// SIMATIC S7-200 project (STEP 7-Micro/WIN), CPU 224XP REL 02.01

SYMBOL_TABLE 用户定义1
TJBZW            M0.3     // 停机标志位
TJ               Q0.7     // 停机
DJD              I0.1     // 电接点压力低
YLD              T45      // 压力低延时
YJQT             I0.5     // 一键启停
GZSC             Q0.5     // 故障输出
ZSGG             M0.1     // 转速过高标志位
Jiansu           Q0.3     // 减速
ZDTS             M0.5     // 自动提速
QDCG             M0.0     // 启动成功位
GF               Q0.6     // 关阀
FMKDW            I0.3     // 阀门开到位
KF               Q0.2     // 开阀
JS               Q0.1     // 加速
YLDXH            M10.0    // 压力低标志位
ZD               I0.0     // 自动
ZDTR             Q0.4     // 自动投入指示
TZ               M10.3    // 停止位
QD               M10.2    // 启动位
END_SYMBOL_TABLE

ORGANIZATION_BLOCK 主程序:OB1
TITLE=程序注释
BEGIN
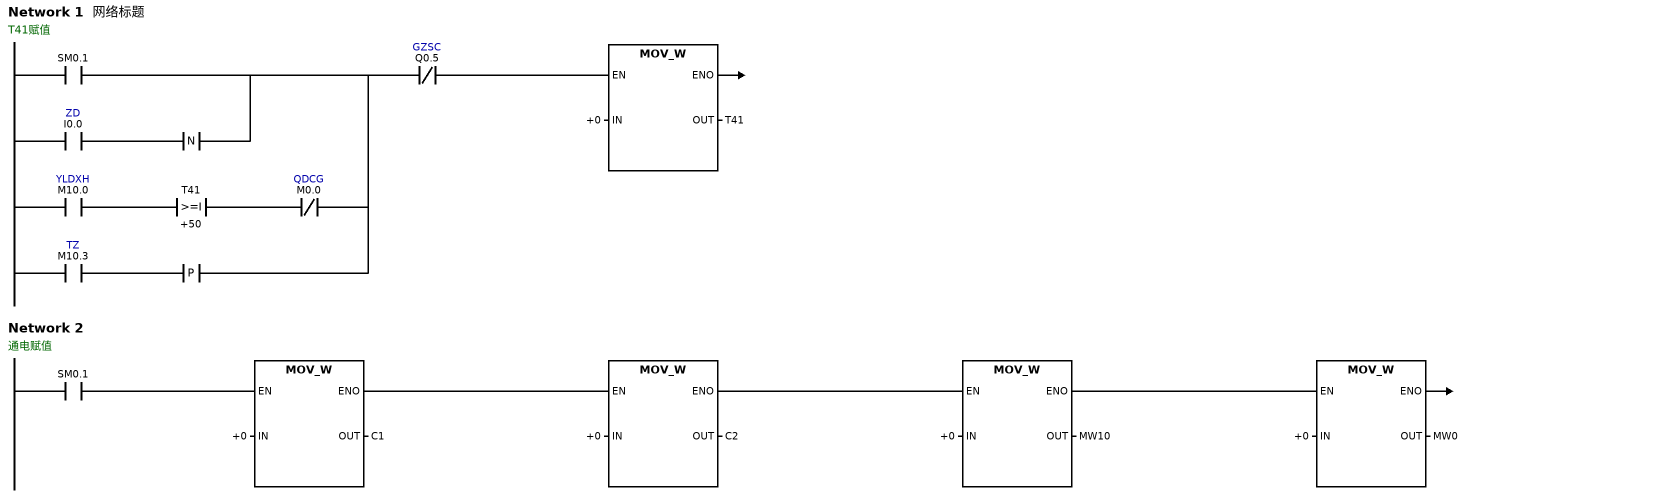
Network 1 // 网络标题
// T41赋值
LD     SM0.1
LD     ZD:I0.0
ED
OLD
LD     YLDXH:M10.0
AW>=   T41, +50
AN     QDCG:M0.0
OLD
LD     TZ:M10.3
EU
OLD
AN     GZSC:Q0.5
MOVW   +0, T41
Network 2
// 通电赋值
LD     SM0.1
MOVW   +0, C1
AENO
MOVW   +0, C2
AENO
MOVW   +0, MW10
AENO
MOVW   +0, MW0
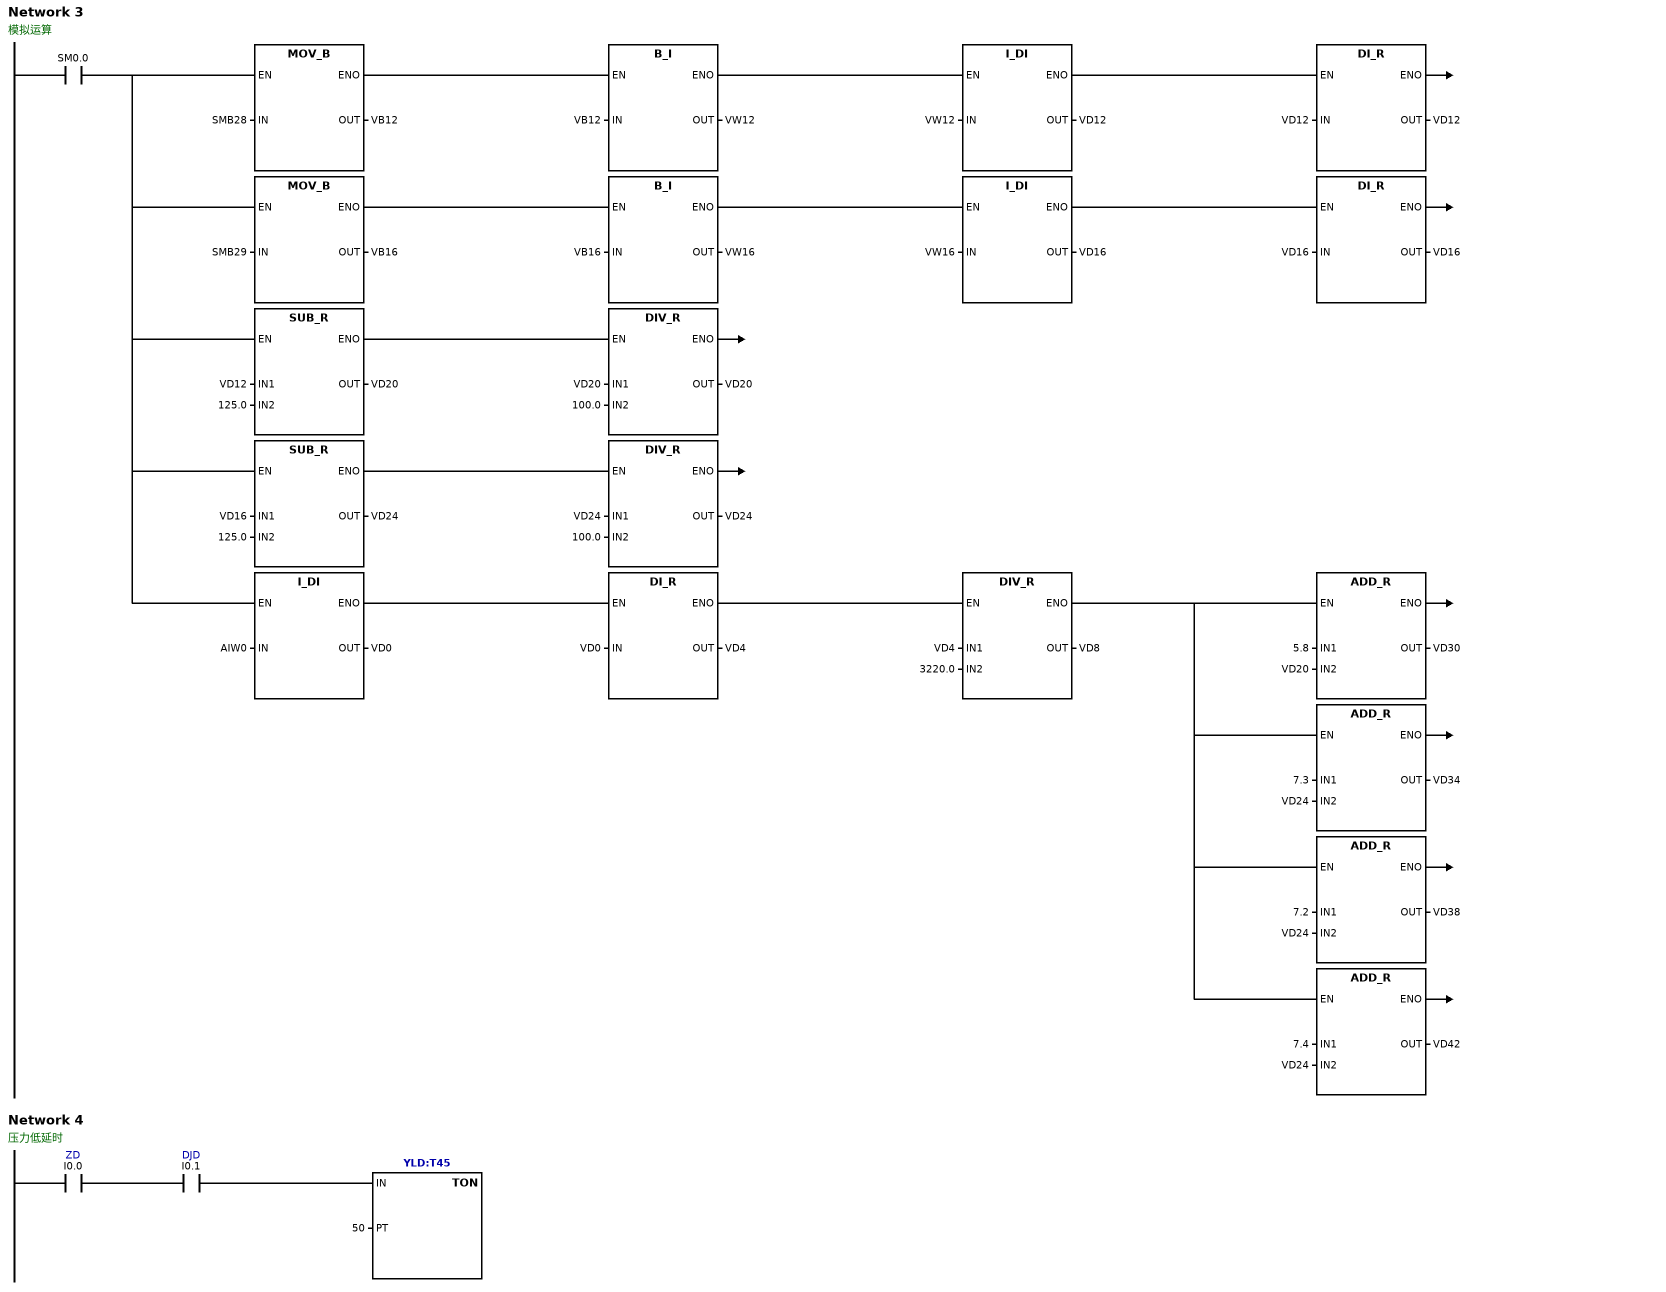
Network 3
// 模拟运算
LD     SM0.0
LPS
MOVB   SMB28, VB12
AENO
BTI    VB12, VW12
AENO
ITD    VW12, VD12
AENO
DTR    VD12, VD12
LRD
MOVB   SMB29, VB16
AENO
BTI    VB16, VW16
AENO
ITD    VW16, VD16
AENO
DTR    VD16, VD16
LRD
MOVR   VD12, VD20
AENO
-R     125.0, VD20
AENO
/R     100.0, VD20
LRD
MOVR   VD16, VD24
AENO
-R     125.0, VD24
AENO
/R     100.0, VD24
LPP
ITD    AIW0, VD0
AENO
DTR    VD0, VD4
AENO
MOVR   VD4, VD8
AENO
/R     3220.0, VD8
AENO
MOVR   5.8, VD30
+R     VD20, VD30
MOVR   7.3, VD34
+R     VD24, VD34
MOVR   7.2, VD38
+R     VD24, VD38
MOVR   7.4, VD42
+R     VD24, VD42
Network 4
// 压力低延时
// (network saved uncompiled; LAD cells follow)
// row 0: c0 -| |- ZD:I0.0  c1 -| |- DJD:I0.1  c2 --  c3 [TON YLD:T45 IN:=power@row0, PT:=50]
// row 1: c3 [box]
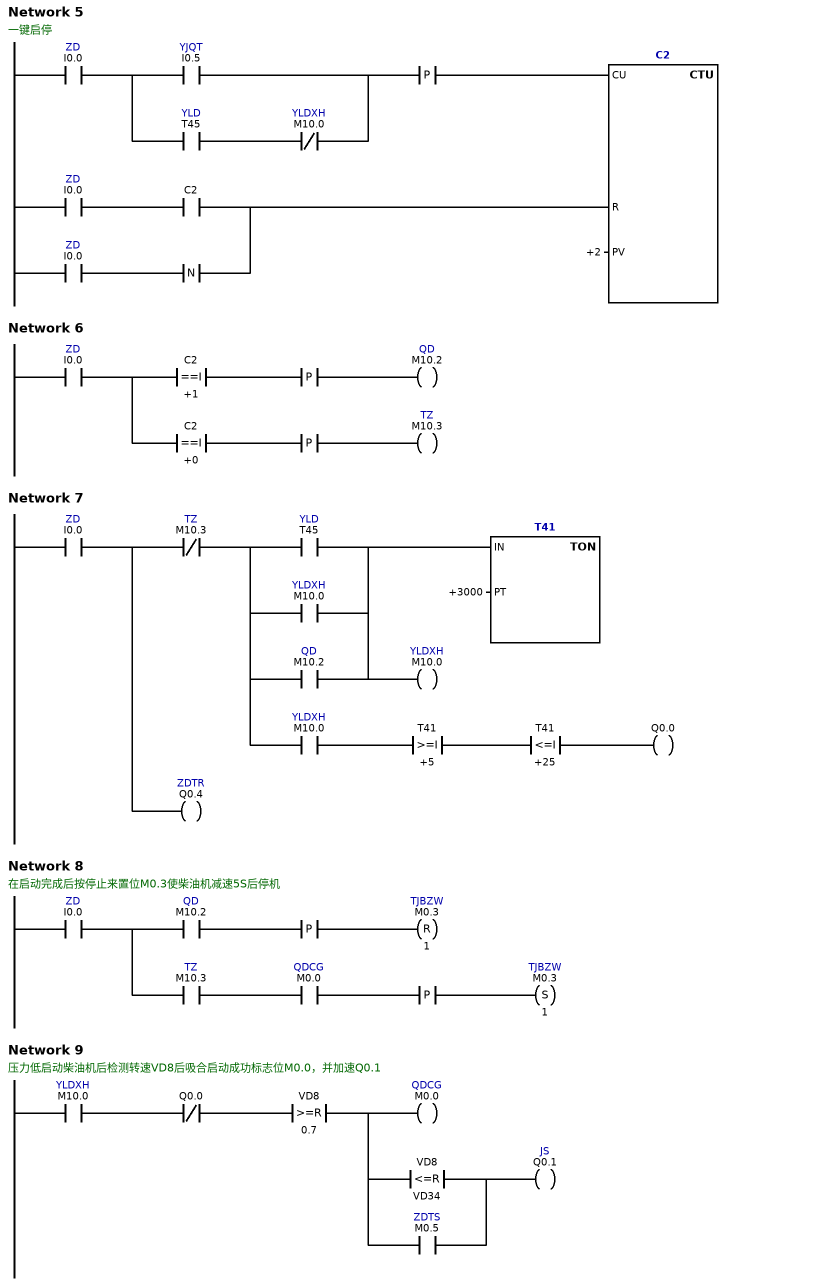
Network 5
// 一键启停
// (network saved uncompiled; LAD cells follow)
// row 0: c0 -| |- ZD:I0.0 v  c1 -| |- YJQT:I0.5  c2 -- v  c3 -|P|-  c4 --  c5 [CTU C2 CU:=power@row0, R:=power@row2, PV:=+2]
// row 1: c0 ^  c1 -| |- YLD:T45  c2 -|/|- YLDXH:M10.0 ^  c5 [box]
// row 2: c0 -| |- ZD:I0.0  c1 -| |- C2 v  c2 --  c3 --  c4 --  c5 [box]
// row 3: c0 -| |- ZD:I0.0  c1 -|N|-  ^  c5 [box]
Network 6
LD     ZD:I0.0
LPS
AW=    C2, +1
EU
=      QD:M10.2
LPP
AW=    C2, +0
EU
=      TZ:M10.3
Network 7
LD     ZD:I0.0
LPS
AN     TZ:M10.3
LPS
LD     YLD:T45
O      YLDXH:M10.0
O      QD:M10.2
ALD
TON    T41, +3000
=      YLDXH:M10.0
LPP
A      YLDXH:M10.0
AW>=   T41, +5
AW<=   T41, +25
=      Q0.0
LPP
=      ZDTR:Q0.4
Network 8
// 在启动完成后按停止来置位M0.3使柴油机减速5S后停机
// (network saved uncompiled; LAD cells follow)
// row 0: c0 -| |- ZD:I0.0 v  c1 -| |- QD:M10.2  c2 -|P|-  c3 -(R) TJBZW:M0.3, 1
// row 1: c0 ^  c1 -| |- TZ:M10.3  c2 -| |- QDCG:M0.0  c3 -|P|-  c4 -(S) TJBZW:M0.3, 1
Network 9
// 压力低启动柴油机后检测转速VD8后吸合启动成功标志位M0.0，并加速Q0.1
LD     YLDXH:M10.0
AN     Q0.0
AR>=   VD8, 0.7
=      QDCG:M0.0
LDR<=  VD8, VD34
O      ZDTS:M0.5
ALD
=      JS:Q0.1
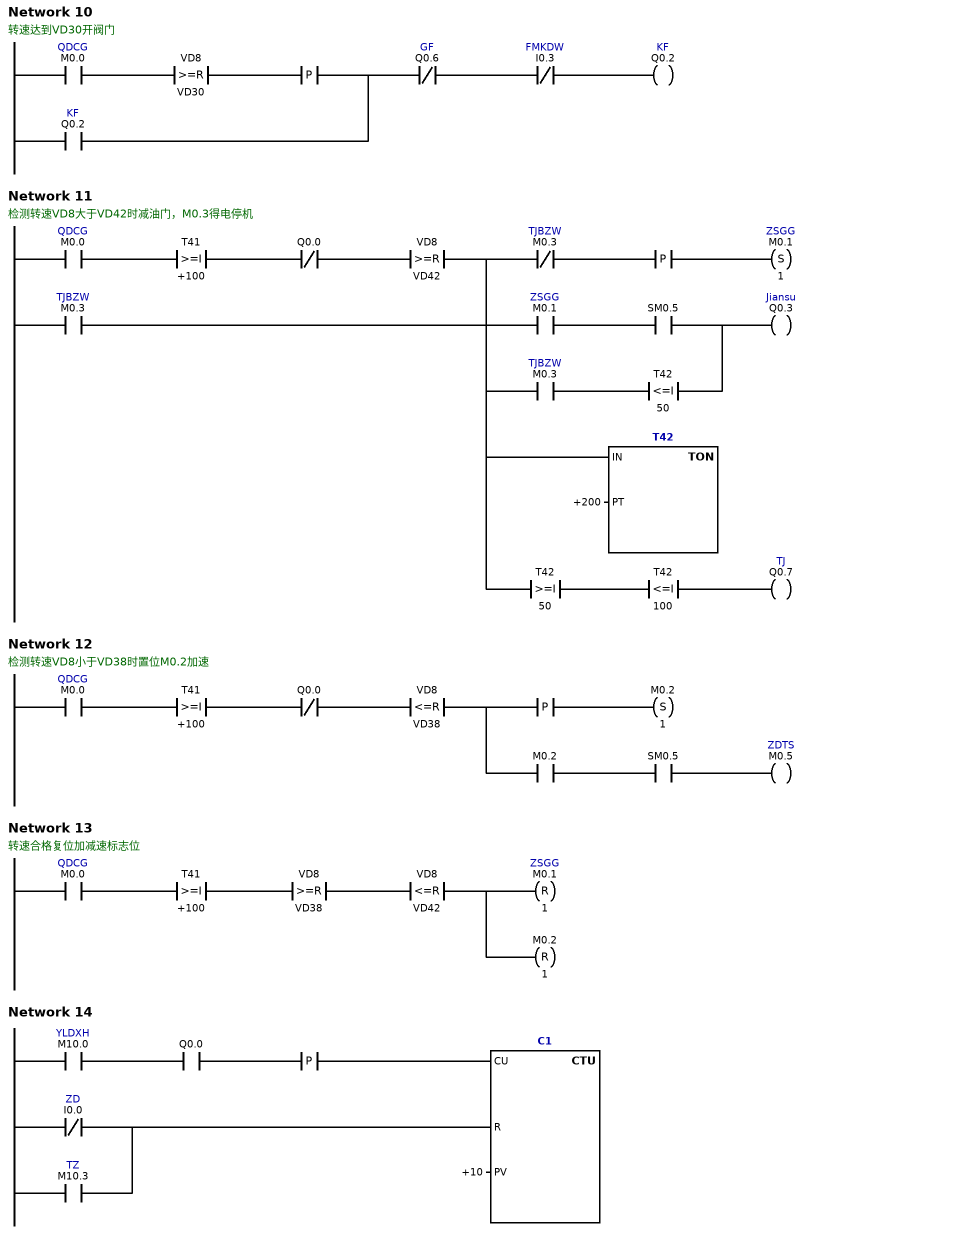
Network 10
// 转速达到VD30开阀门
LD     QDCG:M0.0
AR>=   VD8, VD30
EU
O      KF:Q0.2
AN     GF:Q0.6
AN     FMKDW:I0.3
=      KF:Q0.2
Network 11
// 检测转速VD8大于VD42时减油门，M0.3得电停机
// (network saved uncompiled; LAD cells follow)
// row 0: c0 -| |- QDCG:M0.0  c1 -|>=I|- T41, +100  c2 -|/|- Q0.0  c3 -|>=R|- VD8, VD42 v  c4 -|/|- TJBZW:M0.3  c5 -|P|-  c6 -(S) ZSGG:M0.1, 1
// row 1: c0 -| |- TJBZW:M0.3  c1 --  c2 --  c3 -- ^v  c4 -| |- ZSGG:M0.1  c5 -| |- SM0.5 v  c6 -( ) Jiansu:Q0.3
// row 2: c3 ^v  c4 -| |- TJBZW:M0.3  c5 -|<=I|- T42, 50 ^
// row 3: c3 ^v  c4 --  c5 [TON T42 IN:=power@row3, PT:=+200]
// row 4: c3 ^v  c5 [box]
// row 5: c3 ^  c4 -|>=I|- T42, 50  c5 -|<=I|- T42, 100  c6 -( ) TJ:Q0.7
Network 12
// 检测转速VD8小于VD38时置位M0.2加速
LD     QDCG:M0.0
AW>=   T41, +100
AN     Q0.0
AR<=   VD8, VD38
LPS
EU
S      M0.2, 1
LPP
A      M0.2
A      SM0.5
=      ZDTS:M0.5
Network 13
// 转速合格复位加减速标志位
LD     QDCG:M0.0
AW>=   T41, +100
AR>=   VD8, VD38
AR<=   VD8, VD42
R      ZSGG:M0.1, 1
R      M0.2, 1
Network 14
LD     YLDXH:M10.0
A      Q0.0
EU
LDN    ZD:I0.0
O      TZ:M10.3
CTU    C1, +10
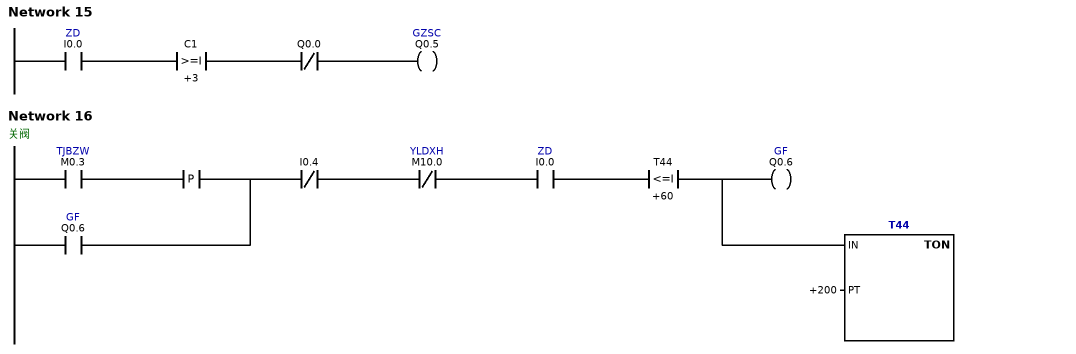
Network 15
LD     ZD:I0.0
AW>=   C1, +3
AN     Q0.0
=      GZSC:Q0.5
Network 16
// 关阀
LD     TJBZW:M0.3
EU
O      GF:Q0.6
AN     I0.4
AN     YLDXH:M10.0
A      ZD:I0.0
AW<=   T44, +60
=      GF:Q0.6
TON    T44, +200
END_ORGANIZATION_BLOCK
